# EPICS autosave request: prosilicaApp/Db/prosilica_settings.req
$(P)$(R)PSReadStatistics.SCAN
$(P)$(R)PSByteRate
$(P)$(R)PSByteRate_RBV.HHSV
$(P)$(R)PSByteRate_RBV.HIGH
$(P)$(R)PSByteRate_RBV.HIHI
$(P)$(R)PSByteRate_RBV.HSV
$(P)$(R)PSByteRate_RBV.LLSV
$(P)$(R)PSByteRate_RBV.LOLO
$(P)$(R)PSByteRate_RBV.LOW
$(P)$(R)PSByteRate_RBV.LSV
$(P)$(R)PSFrameRate_RBV.HHSV
$(P)$(R)PSFrameRate_RBV.HIGH
$(P)$(R)PSFrameRate_RBV.HIHI
$(P)$(R)PSFrameRate_RBV.HSV
$(P)$(R)PSFrameRate_RBV.LLSV
$(P)$(R)PSFrameRate_RBV.LOLO
$(P)$(R)PSFrameRate_RBV.LOW
$(P)$(R)PSFrameRate_RBV.LSV
$(P)$(R)PSFramesCompletedRate_RBV.HHSV
$(P)$(R)PSFramesCompletedRate_RBV.HIGH
$(P)$(R)PSFramesCompletedRate_RBV.HIHI
$(P)$(R)PSFramesCompletedRate_RBV.HSV
$(P)$(R)PSFramesCompletedRate_RBV.LLSV
$(P)$(R)PSFramesCompletedRate_RBV.LOLO
$(P)$(R)PSFramesCompletedRate_RBV.LOW
$(P)$(R)PSFramesCompletedRate_RBV.LSV
$(P)$(R)PSFramesDroppedRate_RBV.HHSV
$(P)$(R)PSFramesDroppedRate_RBV.HIGH
$(P)$(R)PSFramesDroppedRate_RBV.HIHI
$(P)$(R)PSFramesDroppedRate_RBV.HSV
$(P)$(R)PSFramesDroppedRate_RBV.LLSV
$(P)$(R)PSFramesDroppedRate_RBV.LOLO
$(P)$(R)PSFramesDroppedRate_RBV.LOW
$(P)$(R)PSFramesDroppedRate_RBV.LSV
$(P)$(R)PSPacketsErroneousRate_RBV.HHSV
$(P)$(R)PSPacketsErroneousRate_RBV.HIGH
$(P)$(R)PSPacketsErroneousRate_RBV.HIHI
$(P)$(R)PSPacketsErroneousRate_RBV.HSV
$(P)$(R)PSPacketsErroneousRate_RBV.LLSV
$(P)$(R)PSPacketsErroneousRate_RBV.LOLO
$(P)$(R)PSPacketsErroneousRate_RBV.LOW
$(P)$(R)PSPacketsErroneousRate_RBV.LSV
$(P)$(R)PSPacketsMissedRate_RBV.HHSV
$(P)$(R)PSPacketsMissedRate_RBV.HIGH
$(P)$(R)PSPacketsMissedRate_RBV.HIHI
$(P)$(R)PSPacketsMissedRate_RBV.HSV
$(P)$(R)PSPacketsMissedRate_RBV.LLSV
$(P)$(R)PSPacketsMissedRate_RBV.LOLO
$(P)$(R)PSPacketsMissedRate_RBV.LOW
$(P)$(R)PSPacketsMissedRate_RBV.LSV
$(P)$(R)PSPacketsReceivedRate_RBV.HHSV
$(P)$(R)PSPacketsReceivedRate_RBV.HIGH
$(P)$(R)PSPacketsReceivedRate_RBV.HIHI
$(P)$(R)PSPacketsReceivedRate_RBV.HSV
$(P)$(R)PSPacketsReceivedRate_RBV.LLSV
$(P)$(R)PSPacketsReceivedRate_RBV.LOLO
$(P)$(R)PSPacketsReceivedRate_RBV.LOW
$(P)$(R)PSPacketsReceivedRate_RBV.LSV
$(P)$(R)PSPacketsRequestedRate_RBV.HHSV
$(P)$(R)PSPacketsRequestedRate_RBV.HIGH
$(P)$(R)PSPacketsRequestedRate_RBV.HIHI
$(P)$(R)PSPacketsRequestedRate_RBV.HSV
$(P)$(R)PSPacketsRequestedRate_RBV.LLSV
$(P)$(R)PSPacketsRequestedRate_RBV.LOLO
$(P)$(R)PSPacketsRequestedRate_RBV.LOW
$(P)$(R)PSPacketsRequestedRate_RBV.LSV
$(P)$(R)PSPacketsResentRate_RBV.HHSV
$(P)$(R)PSPacketsResentRate_RBV.HIGH
$(P)$(R)PSPacketsResentRate_RBV.HIHI
$(P)$(R)PSPacketsResentRate_RBV.HSV
$(P)$(R)PSPacketsResentRate_RBV.LLSV
$(P)$(R)PSPacketsResentRate_RBV.LOLO
$(P)$(R)PSPacketsResentRate_RBV.LOW
$(P)$(R)PSPacketsResentRate_RBV.LSV
$(P)$(R)PSPacketSize_RBV.HHSV
$(P)$(R)PSPacketSize_RBV.HIGH
$(P)$(R)PSPacketSize_RBV.HIHI
$(P)$(R)PSPacketSize_RBV.HSV
$(P)$(R)PSPacketSize_RBV.LLSV
$(P)$(R)PSPacketSize_RBV.LOLO
$(P)$(R)PSPacketSize_RBV.LOW
$(P)$(R)PSPacketSize_RBV.LSV
$(P)$(R)Strobe1CtlDuration
$(P)$(R)Strobe1Delay
$(P)$(R)Strobe1Duration
$(P)$(R)Strobe1Mode
$(P)$(R)SyncOut1Invert
$(P)$(R)SyncOut1Level
$(P)$(R)SyncOut1Mode
$(P)$(R)SyncOut2Invert
$(P)$(R)SyncOut2Level
$(P)$(R)SyncOut2Mode
$(P)$(R)SyncOut3Invert
$(P)$(R)SyncOut3Level
$(P)$(R)SyncOut3Mode
$(P)$(R)TriggerDelay
$(P)$(R)TriggerEvent
$(P)$(R)TriggerOverlap
